Fanuc KAREL source: ko00051.KL

-- PROVISIONAL review KL for V770-1; original PC SHA256 65d5e4cc3a7d85758d6aa2ce48b267184fa10d028c2628714151625120c06ff6
-- Incomplete behavior may be omitted. Consult companion uncertainty JSON. Do not deploy.
PROGRAM KO00051
%NOLOCKGROUP
BEGIN
  -- UNRESOLVED_PC offsets 5-12; opcodes 9D,23
  -- UNRESOLVED_PC offsets 17-66; opcodes 27,27,49,7E,AD,22,1C,22,31,7E,4A
  -- UNRESOLVED_PC offsets 71-75; opcodes 7F
END KO00051
